PROGRAM Alarms
VAR
END_VAR


//
IF  HydraulicPump.fbHydPump.bFaultThermal THEN
	GVL_Event.aAlarm[1]:=TRUE;
	END_IF
	
IF  UpperPreserDrive.fbUupperPreser.bFault THEN
	GVL_Event.aAlarm[2]:=TRUE;
	END_IF
	
IF Scaling.fbPos.OverRange OR Scaling.fbPos.UnderRange THEN
	GVL_Event.aAlarm[3]:=TRUE;
	END_IF
	
IF NOT.Scaling.PressureAI.Valid THEN
	GVL_Event.aAlarm[4]:=TRUE;
	END_IF

END_PROGRAM

(* stored: Version 1.1.0.1, ProductVersion 3.1.4024.15
   POU Alarms: Id {773151f6-7c44-414a-b82f-b36a8bbe826e}, SpecialFunc None *)
